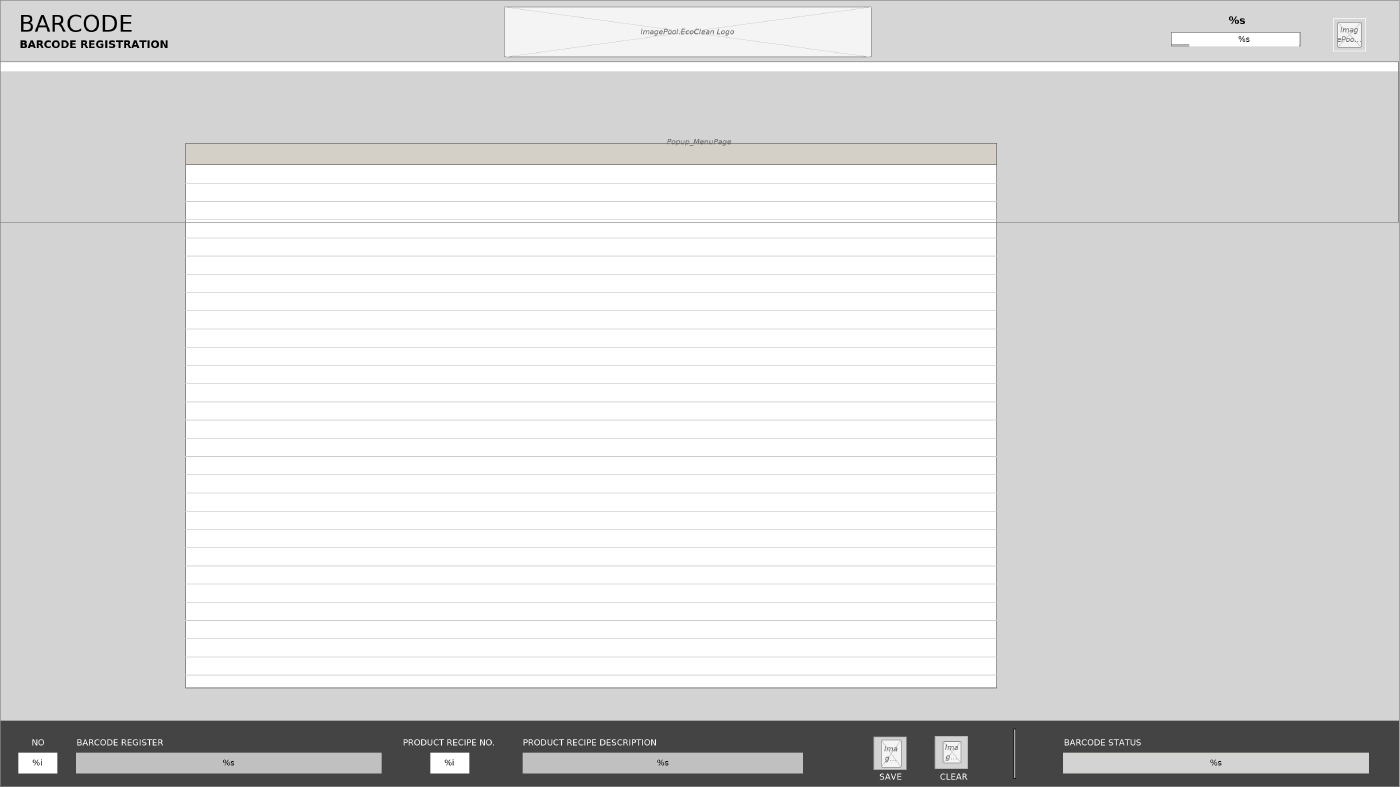
VISUALIZATION Barcode_Page  // 1920x1080
    Rectangle (0,98 1920x981)
    Rectangle (0,63 1920x26)
        p3528305787: HMI_Ctrl.ANIMATION3
    Rectangle (0,0 1919x85)
    Label (23,6 267x53), "BARCODE"
    Label (24,49 320x24), "BARCODE REGISTRATION"
    Rectangle (0,989 1919x91)
    Textfield (1458,1033 419x28), "%s", text variable: Barcode_Reg.sStatus
    Label (1456,1007 127x24), "BARCODE STATUS"
    Rectangle (1390,1000 3x68)
    Textfield (25,1033 53x28), "%i", text variable: iBarcodeRegUserSelectNoDataToSave, input disabled if: iCurrentUserGroupID<3
        OnMouseDown: write the text variable via VisuDialogs.Numpad, min 1, max 100
    Label (26,1007 53x24), "NO"
    Textfield (104,1033 419x28), "%s", text variable: sBarcodeScannerReceivedCmdForReg
    Label (102,1007 413x24), "BARCODE REGISTER"
    Textfield (590,1033 53x28), "%i", text variable: iBarcodeRegUserSelectRecipeNo, input disabled if: iCurrentUserGroupID<3
        OnMouseDown: write the text variable via Default, min 1, max 40
    Label (525,1007 181x24), "PRODUCT RECIPE NO."
    Label (714,1007 387x24), "PRODUCT RECIPE DESCRIPTION"
    Label (1270,1054 76x24), "CLEAR"
    Label (1184,1054 75x24), "SAVE"
    Group (1828,25 45x45)
        OnMouseClick: toggle HMI_Ctrl.MenuButton
        RoundedRectangle (0,0 45x45), colour toggle: HMI_Ctrl.MenuButton
        Image (6,5 33x35), image: ImagePool.Menu Button
    Table (254,196 1113x748), data array: DsAr1sG_BarcodeRegistration
        p3854506369: DsAr1sG_BarcodeRegistration[INDEX].sBarcodeRegistered
        p1892666644: DsAr1sG_BarcodeRegistration[INDEX].iLinkProductRecipeNo
        p338671338: DsAr1sG_BarcodeRegistration[INDEX].bBarcodeRegistrationEn
        p2170511999: DsAr1sG_BarcodeRegistration[INDEX].sLinkProductRecipeDescription
        p2232123230: Barcode Register
        p511219082: Product Recipe
        p4092479075: Product Recipe Description
    Frame (0,84 1918x221), invisible if: HMI_Ctrl.CloseMenuButton
        shows Popup_MenuPage()
    Textfield (717,1033 384x28), "%s", text variable: ARsProductRecipeDescription[iBarcodeRegUserSelectRecipeNo]
    Image (691,9 504x69), image: ImagePool.EcoClean Logo
    Group (1606,17 179x46)
        Button (0,27 177x19), image: VisuSymbols.Symbols.AddUser
        Rectangle (25,28 150x18), "%s", text variable: fbHmiTF1800_UserlevelManagement.dsHmiUserStatus_Active.sLoginName
        Rectangle (2,0 177x22), "%s", text variable: DSLocalSystemTimeML.sCurrentDT24Hr_General
    Group (1198,1011 45x45), input disabled if: bMainOnOff
        RoundedRectangle (0,0 45x45), colour toggle: bBarcodeRegSave
            tap bBarcodeRegSave
        Image (10,4 28x38), image: ImagePool.Save Button
            OnMouseDown: execute { bBarcodeRegSave:=1; }
            OnMouseUp: execute { bBarcodeRegSave:=0; }
    Group (1282,1010 45x45)
        RoundedRectangle (0,0 45x45), colour toggle: bBarcodeRegClear
            tap bBarcodeRegClear
        Image (11,7 25x30), image: ImagePool.Clear Button
            OnMouseDown: execute { bBarcodeRegClear:=1; }
            OnMouseUp: execute { bBarcodeRegClear:=0; }
END_VISUALIZATION

(* stored: Version 1.1.0.1, ProductVersion 3.1.4024.12
   Visu Barcode_Page: Id {28ef272e-9d0a-4bbf-b442-4347d7e22257} *)
